// TIA Portal V20 export
TYPE "HMI_ILck4x3L"
   STRUCT
      In01_Text : String[16];   // In01 text
      BypIn : Word := 16#0;   // Bypass In01 - In08 (via operator) / Bypass In01 (via operator)
      AV01 : Real;   // Analog value for In01
      AV01_Unit : Int := 0;   // Engineering unit of AV01
      In02_Text : String[16];   // In02 text
      AV02 : Real;   // Analog value for In02
      AV02_Unit : Int := 0;   // Engineering unit of AV02
      In03_Text : String[16];   // In03 text
      AV03 : Real;   // Analog value for In03
      AV03_Unit : Int := 0;   // Engineering unit of AV03
      In04_Text : String[16];   // In04 text
      AV04 : Real;   // Analog value for In04
      AV04_Unit : Int := 0;   // Engineering unit of AV04
      In05_Text : String[16];   // In05 text
      AV05 : Real;   // Analog value for In05
      AV05_Unit : Int;   // Engineering unit of AV05
      In06_Text : String[16];   // In06 text
      AV06 : Real;   // Analog value for In06
      AV06_Unit : Int;   // Engineering unit of AV06
      In07_Text : String[16];   // In07 text
      AV07 : Real;   // Analog value for In07
      AV07_Unit : Int;   // Engineering unit of AV07
      In08_Text : String[16];   // In08 text
      AV08 : Real;   // Analog value for In08
      AV08_Unit : Int;   // Engineering unit of AV08
      BypOp : DWord;   // Temp. Bypass by operator In01 - In16, Out
      BypTime : Real := 30.0;   // Temp. Bypass TIME[s]
      BypPreWarnTime : Real := 10.0;   // Temp. Bypass prewarning TIME[s]
      BypRST : Bool;   // Temp. Bypass Restart
      RstOp : Bool := FALSE;   // Reset Interlock by operator
      Out_Byp : Bool;   // Bypass by operator
      RstFirstOp : Bool;   // Reset FirstIn (operator)
      RstBypOp : Bool := FALSE;   // Reset all Bypasses (Operator)
      ILckTime : Real;   // Time on-/off delay or timed Interlock[s]
      BypTime_Out { ExternalWritable := 'False'} : Real;   // Temp. Bypass time left
      ILckTime_Out { ExternalWritable := 'False'} : Real;   // Interlock time left
      OS_PermOut { ExternalWritable := 'False'} : DWord := DWORD#16#FFFF_FFFF;   // Operator Permission: Output for OS
      OS_PermLog { ExternalWritable := 'False'} : DWord := DWORD#16#FFFF_FFFF;   // Operator Permission: Output for OS
      OpSt_Out { ExternalWritable := 'False'} : DWord := 16#0000_0000;   // Enabled operator stations
      TimeMode { ExternalWritable := 'False'} : Int;   // 0: No delay, 1: off delay, 2: on delay, 3: timed (Off), 4: timed (On)
      ST_Worst { ExternalWritable := 'False'} : Byte := 16#80;   // Worst Signal Status
      Out_Word { ExternalWritable := 'False'} : Word;   // Output(Output,Stage 1 - Stage 3)
      AV01_04_ST { ExternalWritable := 'False'} : DWord := DWORD#16#FFFF_FFFF;   // Analog value Signal Status for In01 - In04
      AV05_08_ST { ExternalWritable := 'False'} : DWord := DWORD#16#FFFF_FFFF;   // Analog value Signal Status for In05 - In08
      In01_04_ST { ExternalWritable := 'False'} : DWord := DWORD#16#FFFF_FFFF;   // Signal Status for In01 - In04
      In05_08_ST { ExternalWritable := 'False'} : DWord := DWORD#16#FFFF_FFFF;   // Signal Status for In05 - In08
      Out_ST { ExternalWritable := 'False'} : Byte := BYTE#16#FF;   // Output Signal Status
      Status1 { ExternalWritable := 'False'} : DWord := 16#0000_0000;   // Status1
      Status2 { ExternalWritable := 'False'} : DWord := 16#0000_0000;   // Status2
      Status3 { ExternalWritable := 'False'} : DWord := 16#0000_0000;   // Status3
      Status4 { ExternalWritable := 'False'} : DWord := 16#0000_0000;   // Status4
      Status5 { ExternalWritable := 'False'} : DWord := 16#0000_0000;   // Status5
      Status6 { ExternalWritable := 'False'} : DWord := 16#0000_0000;   // Status6
      Status7 { ExternalWritable := 'False'} : DWord := 16#0000_0000;   // Status7
      Status8 { ExternalWritable := 'False'} : DWord := 16#0000_0000;   // Status8
      Status9 { ExternalWritable := 'False'} : DWord;   // Status9
      Status10 { ExternalWritable := 'False'} : DWord;   // Status10
      Status13 { ExternalWritable := 'False'} : DWord;   // Status13
   END_STRUCT;
END_TYPE
